(* PLC project Tc2_Utilities.ULARGE_TO_ULINT Demo, tc3-libraries-kb TwinCAT 3.1 *)
(* stored: creationDateTime 2026-05-10T18:00:00, modificationDateTime 2026-05-10T18:00:00 *)

PROGRAM P_Demo_ULARGE_TO_ULINT
  VAR
    rResult : ULINT;  (* ULARGE_TO_ULINT 返回值 *)
    bRun : BOOL;  (* 触发一次调用 *)
    tu : T_ULARGE_INTEGER;  (* 测试用本地变量 *)
  END_VAR

            // ============================================================
// Tc2_Utilities.ULARGE_TO_ULINT 演示程序（FUNCTION）
// ============================================================
// 验证步骤：
//   1. 引用 Tc2_Utilities
//   2. 编译 + 登录
//   3. 强制 bRun := TRUE 一个周期
//   4. 在线监视 rResult
// ============================================================

tu := ULARGE_INTEGER(0, 100);
IF bRun THEN
    rResult := ULARGE_TO_ULINT(tu);
    bRun := FALSE;
END_IF;

          
END_PROGRAM
